// Mitsubishi GX Works2 project: 1008최신화   PLC: Q02U

PROGRAM INPUT
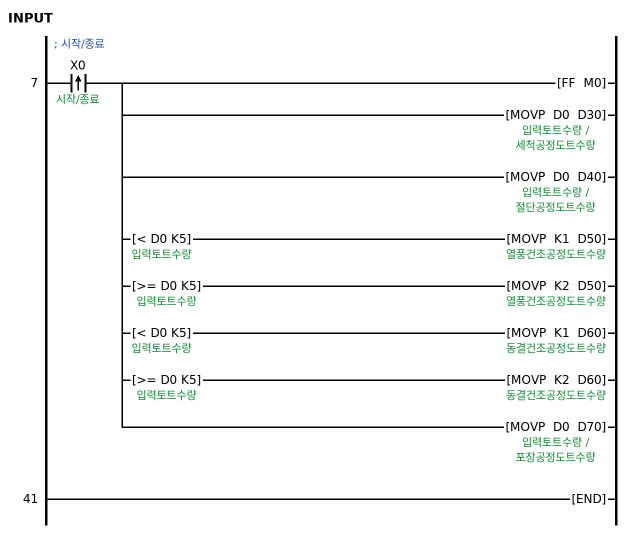
; 시작/종료
7     LDP     X0  ; 시작/종료
      FF      M0
      MOVP    D0 D30  ; 입력토트수량 / 세척공정도트수량
      MOVP    D0 D40  ; 절단공정도트수량
      MPS
      AND<    D0 K5  ; 입력토트수량
      MOVP    K1 D50  ; 열풍건조공정도트수량
      MRD
      AND>=   D0 K5  ; 입력토트수량
      MOVP    K2 D50
      MRD
      AND<    D0 K5  ; 입력토트수량
      MOVP    K1 D60  ; 동결건조공정도트수량
      MRD
      AND>=   D0 K5  ; 입력토트수량
      MOVP    K2 D60
      MPP
      MOVP    D0 D70  ; 포장공정도트수량
41    END
END_PROGRAM

PROGRAM 세척공정
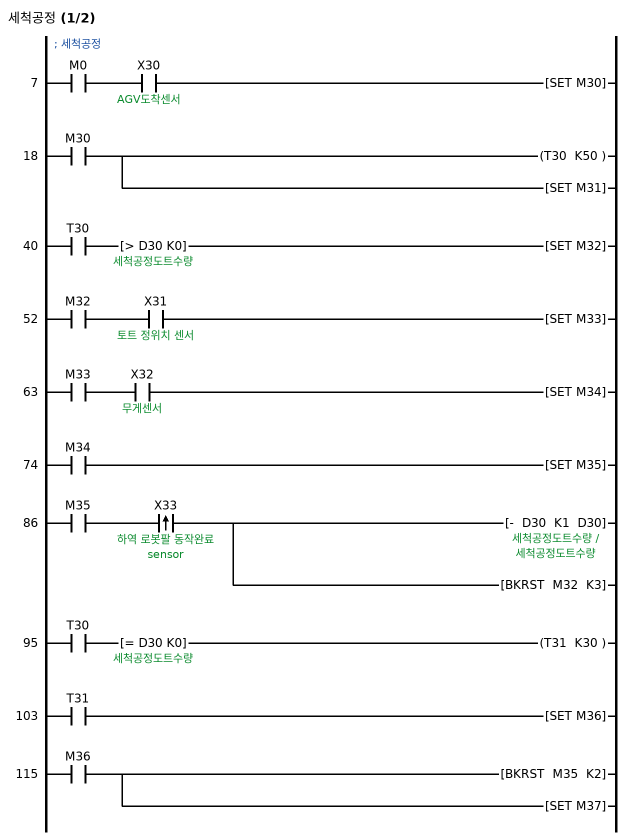
; 세척공정
7     LD      M0
      AND     X30  ; AGV도착센서
      SET     M30
        [note] 펌프모터 ON
18    LD      M30
      OUT     T30 K50
        [note] 펌핑모터 OFF
      SET     M31
        [note] SubCVY ON
40    LD      T30
      AND>    D30 K0  ; 세척공정도트수량
      SET     M32
        [note] 토트 발생
52    LD      M32
      AND     X31  ; 토트 정위치 센서
      SET     M33
        [note] MainCVY ON
63    LD      M33
      AND     X32  ; 무게센서
      SET     M34
        [note] MainCVY OFF
74    LD      M34
      SET     M35
        [note] 하역 로봇팔 ON
86    LD      M35
      ANDP    X33  ; 하역 로봇팔 동작완료 sensor
      -       D30 K1 D30
      BKRST   M32 K3
95    LD      T30
      AND=    D30 K0  ; 세척공정도트수량
      OUT     T31 K30
103   LD      T31
      SET     M36
        [note] 하역 로봇팔 OFF
115   LD      M36
      BKRST   M35 K2
      SET     M37
        [note] AGV 다음 공정 이동, SubCVY OFF
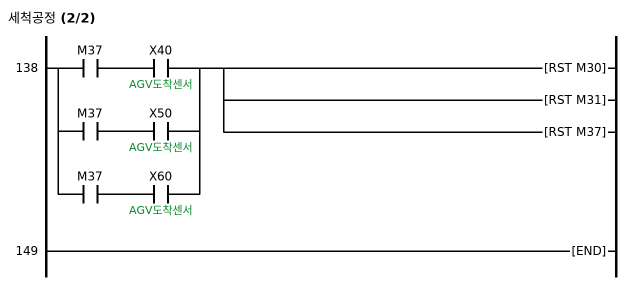
138   LD      M37
      AND     X40  ; AGV도착센서
      LD      M37
      AND     X50  ; AGV도착센서
      ORB
      LD      M37
      AND     X60  ; AGV도착센서
      ORB
      RST     M30
      RST     M31
      RST     M37
149   END
END_PROGRAM

PROGRAM 열풍건조
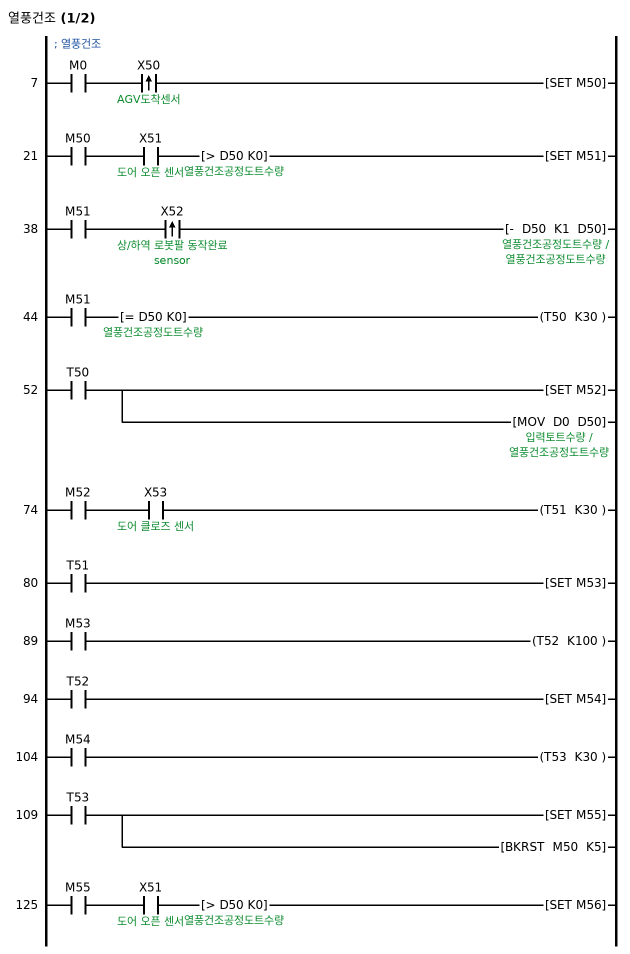
; 열풍건조
7     LD      M0
      ANDP    X50  ; AGV도착센서
      SET     M50
        [note] 도어 오픈모터(정)
21    LD      M50
      AND     X51  ; 도어 오픈 센서
      AND>    D50 K0  ; 열풍건조공정도트수량
      SET     M51
        [note] 상역 로봇 팔동작
38    LD      M51
      ANDP    X52  ; 상/하역 로봇팔 동작완료 sensor
      -       D50 K1 D50
44    LD      M51
      AND=    D50 K0  ; 열풍건조공정도트수량
      OUT     T50 K30
52    LD      T50
      SET     M52
        [note] 도어 클로즈모터(역), 로봇팔 OFF
      MOV     D0 D50  ; 입력토트수량
74    LD      M52
      AND     X53  ; 도어 클로즈 센서
      OUT     T51 K30
80    LD      T51
      SET     M53
        [note] 건조기 ON
89    LD      M53
      OUT     T52 K100
94    LD      T52
      SET     M54
        [note] 건조기 OFF
104   LD      M54
      OUT     T53 K30
109   LD      T53
      SET     M55
        [note] 도어 오픈모터(정)
      BKRST   M50 K5
125   LD      M55
      AND     X51  ; 도어 오픈 센서
      AND>    D50 K0  ; 열풍건조공정도트수량
      SET     M56
        [note] 하역 로봇팔 동작
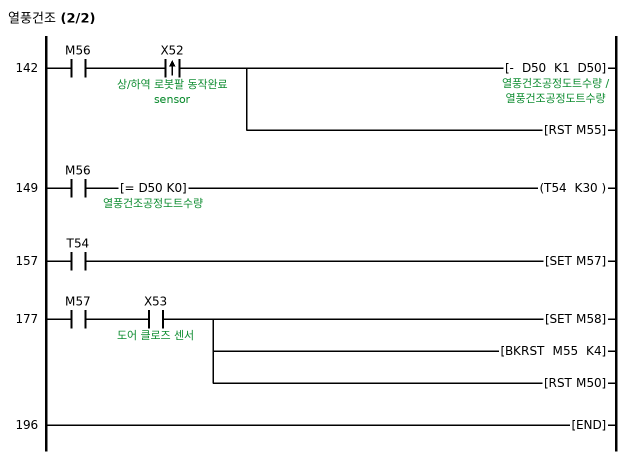
142   LD      M56
      ANDP    X52  ; 상/하역 로봇팔 동작완료 sensor
      -       D50 K1 D50
      RST     M55
149   LD      M56
      AND=    D50 K0  ; 열풍건조공정도트수량
      OUT     T54 K30
157   LD      T54
      SET     M57
        [note] 도어 클로즈모터(역), 로봇팔 OFF
177   LD      M57
      AND     X53  ; 도어 클로즈 센서
      SET     M58
        [note] AGV 다음 공정 이동
      BKRST   M55 K4
      RST     M50
196   END
END_PROGRAM

PROGRAM OUTPUT
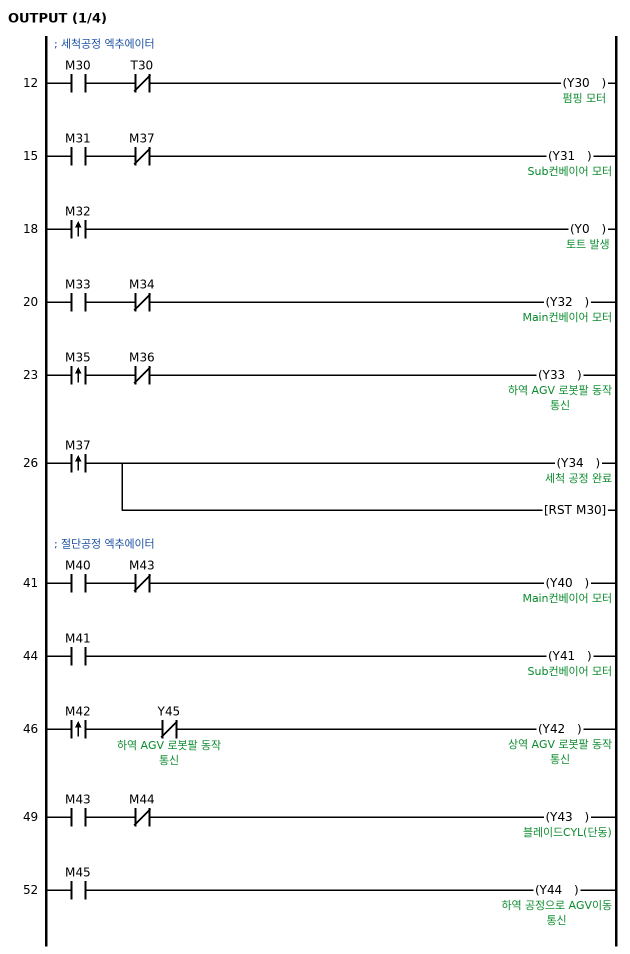
; 세척공정 엑추에이터
12    LD      M30
      ANI     T30
      OUT     Y30  ; 펌핑 모터
15    LD      M31
      ANI     M37
      OUT     Y31  ; Sub컨베이어 모터
18    LDP     M32
      OUT     Y0  ; 토트 발생
20    LD      M33
      ANI     M34
      OUT     Y32  ; Main컨베이어 모터
23    LDP     M35
      ANI     M36
      OUT     Y33  ; 하역 AGV 로봇팔 동작 통신
26    LDP     M37
      OUT     Y34  ; 세척 공정 완료
      RST     M30
; 절단공정 엑추에이터
41    LD      M40
      ANI     M43
      OUT     Y40  ; Main컨베이어 모터
44    LD      M41
      OUT     Y41  ; Sub컨베이어 모터
46    LDP     M42
      ANI     Y45  ; 하역 AGV 로봇팔 동작 통신
      OUT     Y42  ; 상역 AGV 로봇팔 동작 통신
49    LD      M43
      ANI     M44
      OUT     Y43  ; 블레이드CYL(단동)
52    LD      M45
      OUT     Y44  ; 하역 공정으로 AGV이동 통신
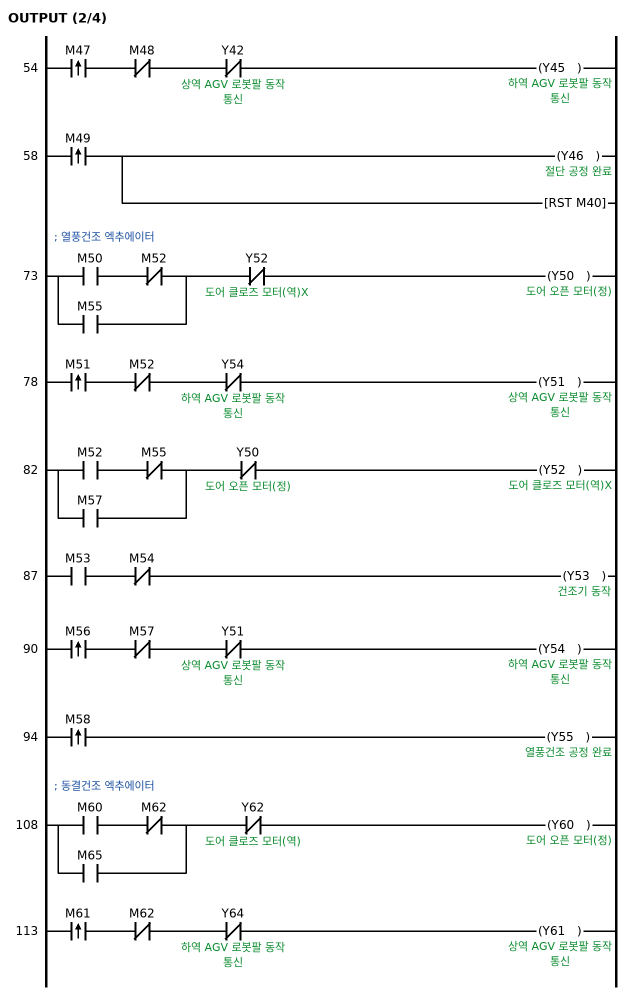
54    LDP     M47
      ANI     M48
      ANI     Y42  ; 상역 AGV 로봇팔 동작 통신
      OUT     Y45  ; 하역 AGV 로봇팔 동작 통신
58    LDP     M49
      OUT     Y46  ; 절단 공정 완료
      RST     M40
; 열풍건조 엑추에이터
73    LD      M50
      ANI     M52
      OR      M55
      ANI     Y52  ; 도어 클로즈 모터(역)X
      OUT     Y50  ; 도어 오픈 모터(정)
78    LDP     M51
      ANI     M52
      ANI     Y54  ; 하역 AGV 로봇팔 동작 통신
      OUT     Y51  ; 상역 AGV 로봇팔 동작 통신
82    LD      M52
      ANI     M55
      OR      M57
      ANI     Y50  ; 도어 오픈 모터(정)
      OUT     Y52  ; 도어 클로즈 모터(역)X
87    LD      M53
      ANI     M54
      OUT     Y53  ; 건조기 동작
90    LDP     M56
      ANI     M57
      ANI     Y51  ; 상역 AGV 로봇팔 동작 통신
      OUT     Y54  ; 하역 AGV 로봇팔 동작 통신
94    LDP     M58
      OUT     Y55  ; 열풍건조 공정 완료
; 동결건조 엑추에이터
108   LD      M60
      ANI     M62
      OR      M65
      ANI     Y62  ; 도어 클로즈 모터(역)
      OUT     Y60  ; 도어 오픈 모터(정)
113   LDP     M61
      ANI     M62
      ANI     Y64  ; 하역 AGV 로봇팔 동작 통신
      OUT     Y61  ; 상역 AGV 로봇팔 동작 통신
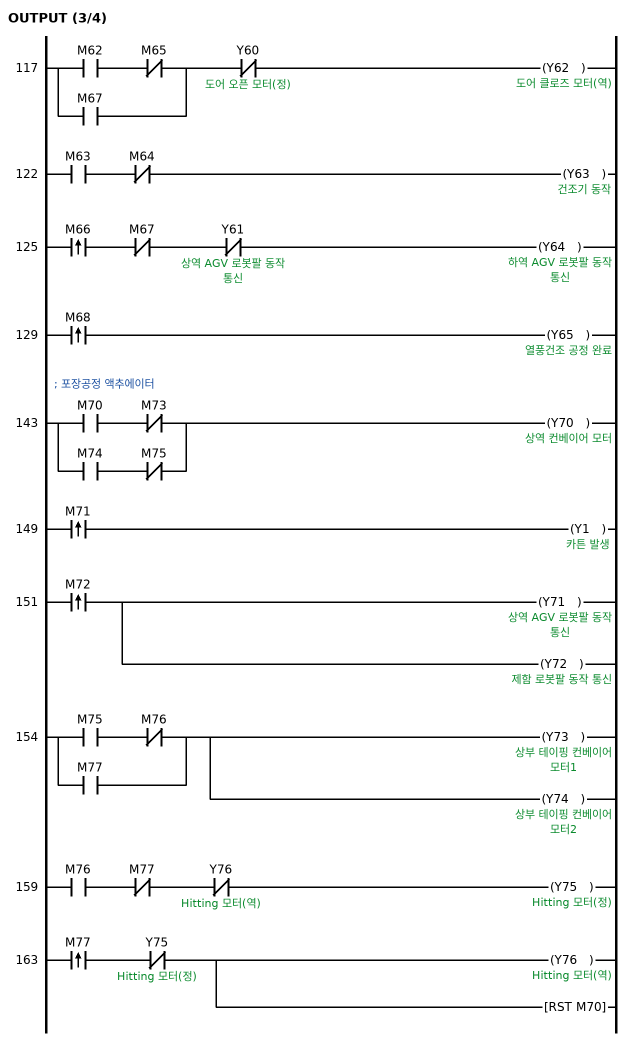
117   LD      M62
      ANI     M65
      OR      M67
      ANI     Y60  ; 도어 오픈 모터(정)
      OUT     Y62  ; 도어 클로즈 모터(역)
122   LD      M63
      ANI     M64
      OUT     Y63  ; 건조기 동작
125   LDP     M66
      ANI     M67
      ANI     Y61  ; 상역 AGV 로봇팔 동작 통신
      OUT     Y64  ; 하역 AGV 로봇팔 동작 통신
129   LDP     M68
      OUT     Y65  ; 열풍건조 공정 완료
; 포장공정 액추에이터
143   LD      M70
      ANI     M73
      LD      M74
      ANI     M75
      ORB
      OUT     Y70  ; 상역 컨베이어 모터
149   LDP     M71
      OUT     Y1  ; 카튼 발생
151   LDP     M72
      OUT     Y71  ; 상역 AGV 로봇팔 동작 통신
      OUT     Y72  ; 제함 로봇팔 동작 통신
154   LD      M75
      ANI     M76
      OR      M77
      OUT     Y73  ; 상부 테이핑 컨베이어 모터1
      OUT     Y74  ; 상부 테이핑 컨베이어 모터2
159   LD      M76
      ANI     M77
      ANI     Y76  ; Hitting 모터(역)
      OUT     Y75  ; Hitting 모터(정)
163   LDP     M77
      ANI     Y75  ; Hitting 모터(정)
      OUT     Y76  ; Hitting 모터(역)
      RST     M70
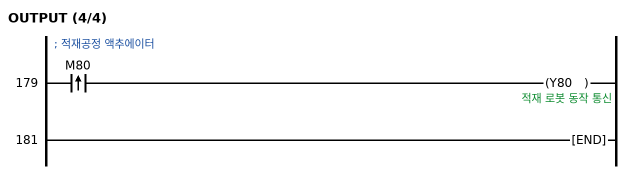
; 적재공정 액추에이터
179   LDP     M80
      OUT     Y80  ; 적재 로봇 동작 통신
181   END
END_PROGRAM

PROGRAM 동결건조
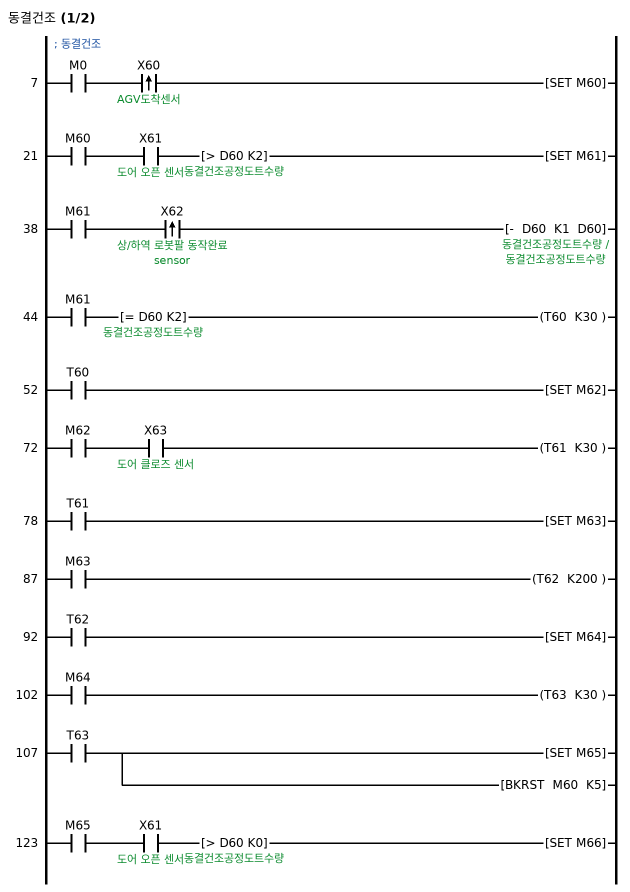
; 동결건조
7     LD      M0
      ANDP    X60  ; AGV도착센서
      SET     M60
        [note] 도어 오픈모터(정)
21    LD      M60
      AND     X61  ; 도어 오픈 센서
      AND>    D60 K2  ; 동결건조공정도트수량
      SET     M61
        [note] 상역 로봇 팔동작
38    LD      M61
      ANDP    X62  ; 상/하역 로봇팔 동작완료 sensor
      -       D60 K1 D60
44    LD      M61
      AND=    D60 K2  ; 동결건조공정도트수량
      OUT     T60 K30
52    LD      T60
      SET     M62
        [note] 도어 클로즈모터(역), 로봇팔 OFF
72    LD      M62
      AND     X63  ; 도어 클로즈 센서
      OUT     T61 K30
78    LD      T61
      SET     M63
        [note] 건조기 ON
87    LD      M63
      OUT     T62 K200
92    LD      T62
      SET     M64
        [note] 건조기 OFF
102   LD      M64
      OUT     T63 K30
107   LD      T63
      SET     M65
        [note] 도어 오픈모터(정)
      BKRST   M60 K5
123   LD      M65
      AND     X61  ; 도어 오픈 센서
      AND>    D60 K0  ; 동결건조공정도트수량
      SET     M66
        [note] 하역 로봇팔 동작
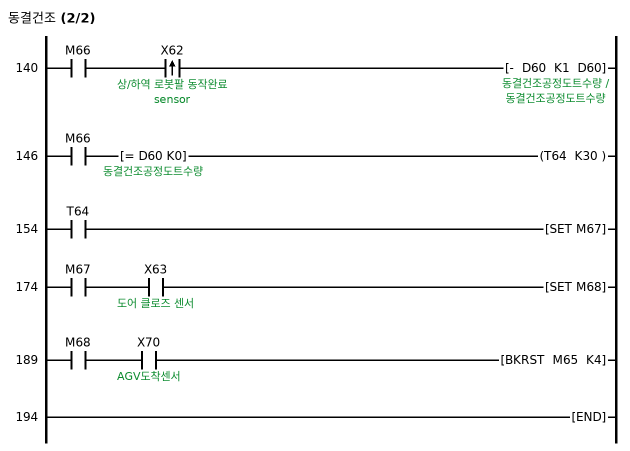
140   LD      M66
      ANDP    X62  ; 상/하역 로봇팔 동작완료 sensor
      -       D60 K1 D60
146   LD      M66
      AND=    D60 K0  ; 동결건조공정도트수량
      OUT     T64 K30
154   LD      T64
      SET     M67
        [note] 도어 클로즈모터(역), 로봇팔 OFF
174   LD      M67
      AND     X63  ; 도어 클로즈 센서
      SET     M68
        [note] AGV 다음 공정 이동
189   LD      M68
      AND     X70  ; AGV도착센서
      BKRST   M65 K4
194   END
END_PROGRAM

PROGRAM 절단공정
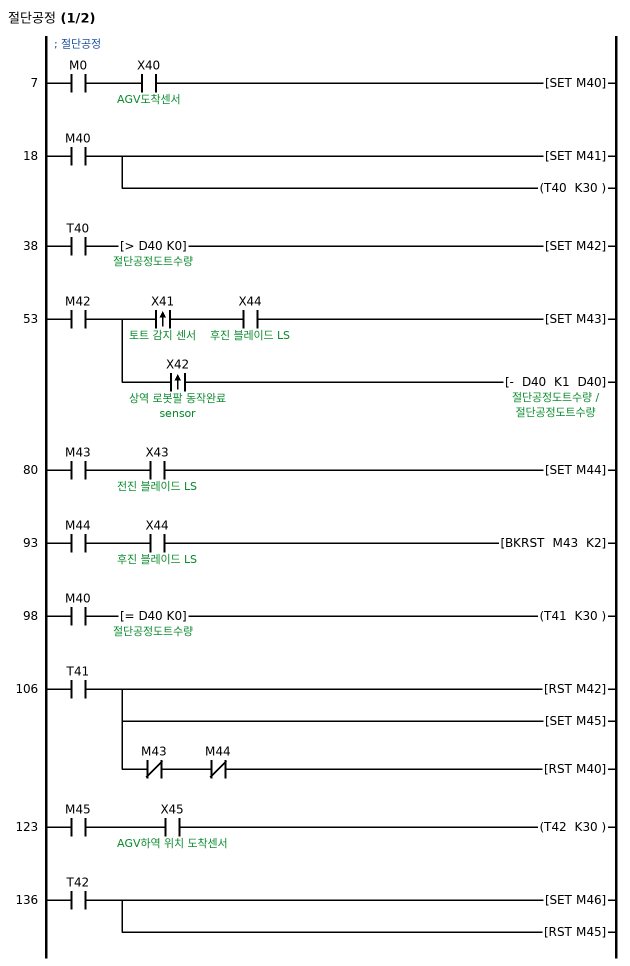
; 절단공정
7     LD      M0
      AND     X40  ; AGV도착센서
      SET     M40
        [note] MainCVY ON
18    LD      M40
      SET     M41
        [note] SubCVY ON
      OUT     T40 K30
        [note] 상역 여유
38    LD      T40
      AND>    D40 K0  ; 절단공정도트수량
      SET     M42
        [note] 상역 로봇팔 ON
53    LD      M42
      MPS
      ANDP    X41  ; 토트 감지 센서
      AND     X44  ; 후진 블레이드 LS
      SET     M43
        [note] MainCVY OFF, 블레이드CYL ON
      MPP
      ANDP    X42  ; 상역 로봇팔 동작완료 sensor
      -       D40 K1 D40
80    LD      M43
      AND     X43  ; 전진 블레이드 LS
      SET     M44
        [note] 블레이드CYL OFF
93    LD      M44
      AND     X44  ; 후진 블레이드 LS
      BKRST   M43 K2
98    LD      M40
      AND=    D40 K0  ; 절단공정도트수량
      OUT     T41 K30
106   LD      T41
      RST     M42
      SET     M45
        [note] AGV하역 위치 이동
      ANI     M43
      ANI     M44
      RST     M40
123   LD      M45
      AND     X45  ; AGV하역 위치 도착센서
      OUT     T42 K30
        [note] 하역 여유
136   LD      T42
      SET     M46
      RST     M45
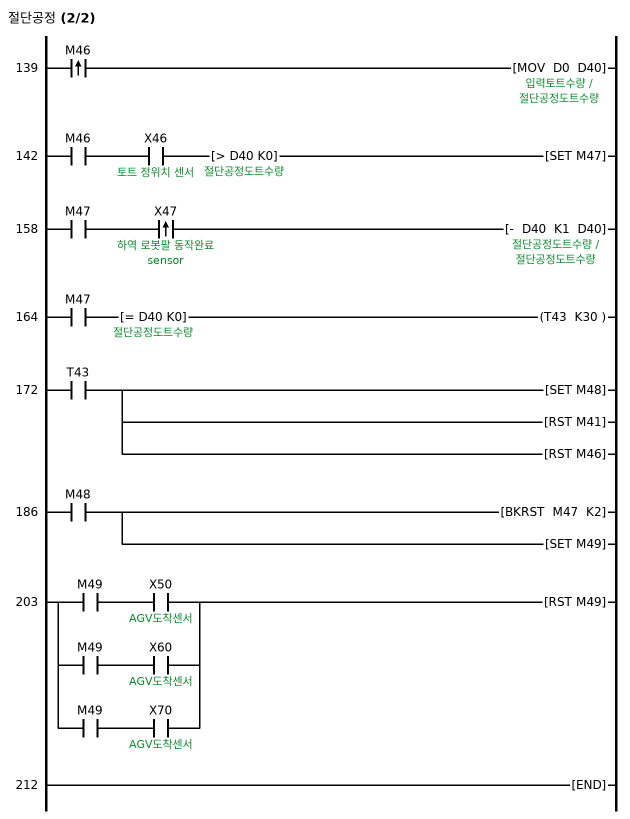
139   LDP     M46
      MOV     D0 D40  ; 입력토트수량
142   LD      M46
      AND     X46  ; 토트 정위치 센서
      AND>    D40 K0  ; 절단공정도트수량
      SET     M47
        [note] 하역 로봇팔 ON
158   LD      M47
      ANDP    X47  ; 하역 로봇팔 동작완료 sensor
      -       D40 K1 D40
164   LD      M47
      AND=    D40 K0  ; 절단공정도트수량
      OUT     T43 K30
172   LD      T43
      SET     M48
        [note] 하역 로봇팔 OFF
      RST     M41
      RST     M46
186   LD      M48
      BKRST   M47 K2
      SET     M49
        [note] AGV 다음 공정 이동
203   LD      M49
      AND     X50  ; AGV도착센서
      LD      M49
      AND     X60  ; AGV도착센서
      ORB
      LD      M49
      AND     X70  ; AGV도착센서
      ORB
      RST     M49
212   END
END_PROGRAM

PROGRAM 포장공정
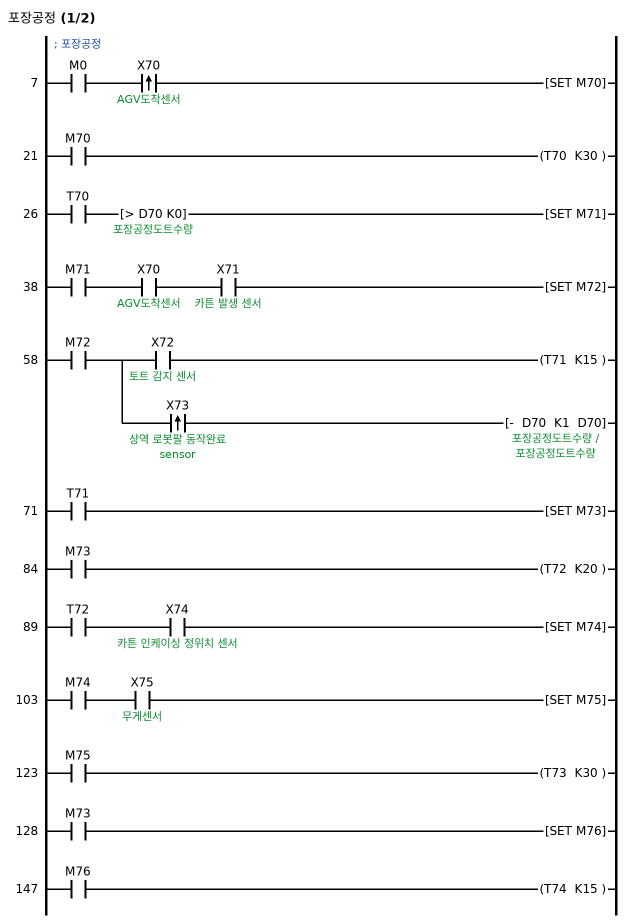
; 포장공정
7     LD      M0
      ANDP    X70  ; AGV도착센서
      SET     M70
        [note] 상역 컨베이어 ON
21    LD      M70
      OUT     T70 K30
26    LD      T70
      AND>    D70 K0  ; 포장공정도트수량
      SET     M71
        [note] 카튼 발생
38    LD      M71
      AND     X70  ; AGV도착센서
      AND     X71  ; 카튼 발생 센서
      SET     M72
        [note] 상역 로봇팔, 제함 로봇팔 ON
58    LD      M72
      MPS
      AND     X72  ; 토트 감지 센서
      OUT     T71 K15
      MPP
      ANDP    X73  ; 상역 로봇팔 동작완료 sensor
      -       D70 K1 D70
71    LD      T71
      SET     M73
        [note] 상역 컨베이어 OFF
84    LD      M73
      OUT     T72 K20
89    LD      T72
      AND     X74  ; 카튼 인케이싱 정위치 센서
      SET     M74
        [note] 상역 컨벤이어 ON
103   LD      M74
      AND     X75  ; 무게센서
      SET     M75
        [note] 상부테이핑CVY ON,상역CVY OFF
123   LD      M75
      OUT     T73 K30
128   LD      M73
      SET     M76
        [note] 상부테이핑CVY OFF, Hitting ON
147   LD      M76
      OUT     T74 K15
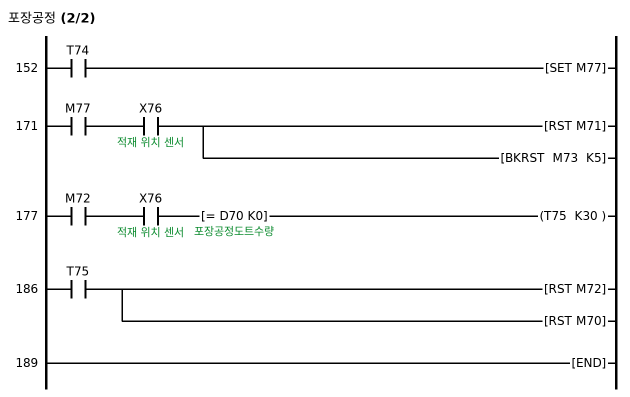
152   LD      T74
      SET     M77
        [note] 상부테이핑CVY ON, Hitting OFF
171   LD      M77
      AND     X76  ; 적재 위치 센서
      RST     M71
      BKRST   M73 K5
177   LD      M72
      AND     X76  ; 적재 위치 센서
      AND=    D70 K0  ; 포장공정도트수량
      OUT     T75 K30
186   LD      T75
      RST     M72
      RST     M70
189   END
END_PROGRAM

PROGRAM 적재공정
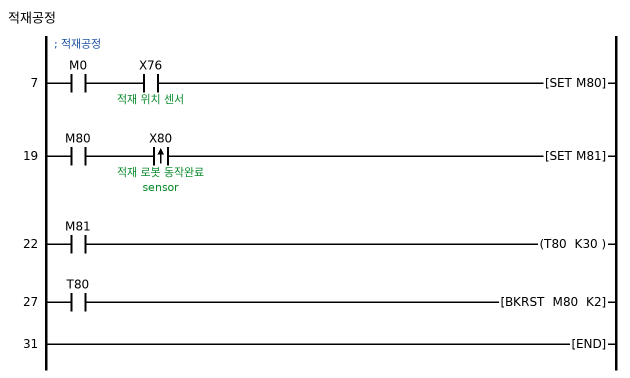
; 적재공정
7     LD      M0
      AND     X76  ; 적재 위치 센서
      SET     M80
        [note] 적재 로봇 ON
19    LD      M80
      ANDP    X80  ; 적재 로봇 동작완료 sensor
      SET     M81
22    LD      M81
      OUT     T80 K30
27    LD      T80
      BKRST   M80 K2
31    END
END_PROGRAM
